// TIA Portal V17 export
// export: Created 2024-10-17T14:16:17.2229745Z, ExportSetting WithDefaults, DisplayName Totally Integrated Automation Portal, DisplayVersion V17 Update 4, DisplayName TIA Portal Openness, DisplayVersion V17 Update 4, DisplayName TIA Portal Version Control Interface, DisplayVersion V17, DisplayName SINAMICS Startdrive Advanced, DisplayVersion V17 Update2, DisplayName SINAMICS Startdrive G130, G150, S120, S150, SINAMICS MV, S210, DisplayVersion V17 Update2, DisplayName SINAMICS Startdrive G110M, G120, G120C, G120D, G120P, G115D, DisplayVersion V17 Update2, DisplayName STEP 7 Professional, DisplayVersion V17 Update 4, DisplayName STEP 7 Safety, DisplayVersion V17, DisplayName WinCC Advanced / Unified PC, DisplayVersion V17 Update 4
TYPE "LPMLV2022_typeCommandIngredients"
TITLE = LPMLV2022_typeCommandIngredients
// Support: tech.team.motioncontrol@siemens.com
// stored: IsFailsafeCompliant false
   STRUCT
      Parameter_REAL : Array[0.."LPMLV2022_COMMAND_INGREDIENTS_PARAMETER_REAL_UPPER_LIM"] of "LPMLV2022_typeParameter_REAL";   // Structured Array of Ingredient information for values with REAL data type
      Parameter_STRING : Array[0.."LPMLV2022_COMMAND_INGREDIENTS_PARAMETER_STRING_UPPER_LIM"] of "LPMLV2022_typeParameter_STRING";   // Structured Array of Ingredient information for values with STRING data type
      Parameter_LREAL : Array[0.."LPMLV2022_COMMAND_INGREDIENTS_PARAMETER_LREAL_UPPER_LIM"] of "LPMLV2022_typeParameter_LREAL";   // Structured Array of Ingredient information for values with LREAL data type
      Parameter_DINT : Array[0.."LPMLV2022_COMMAND_INGREDIENTS_PARAMETER_DINT_UPPER_LIM"] of "LPMLV2022_typeParameter_DINT";   // Structured Array of Ingredient Information for values with DINT data type
      Parameter_BOOL : Array[0.."LPMLV2022_COMMAND_INGREDIENTS_PARAMETER_BOOL_UPPER_LIM"] of "LPMLV2022_typeParameter_BOOL";   // Structured Array of Ingredient Information for values with BOOL data type
   END_STRUCT;
END_TYPE
